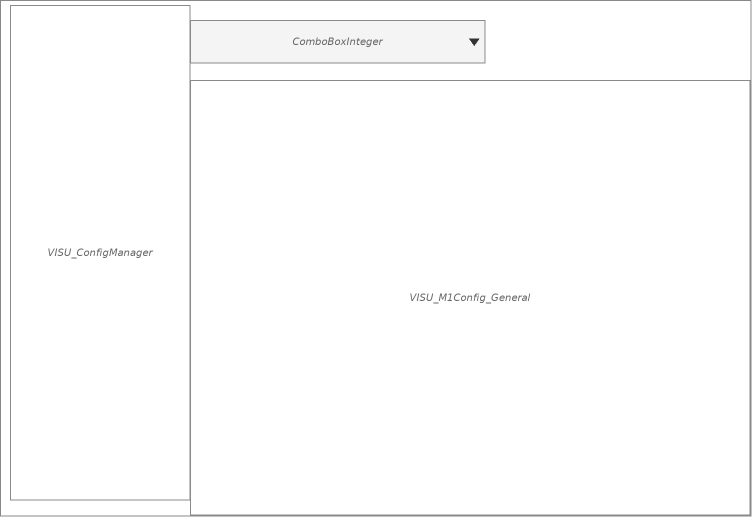
VISUALIZATION VISU_M1Config  // 752x517
VAR_IN_OUT
    editableConfig : M1Config;
	activeConfig : M1Config;
    mgr : ConfigManager;
    mgrWidget : ConfigManagerWidget;
    activeTab : INT;
END_VAR
    Frame (10,5 180x495)
        shows VISU_ConfigManager(mgr := mgr, widget := mgrWidget)
    ComboBoxInteger (190,20 295x43), variable: activeTab, text list: 'M1ConfigTabsTextList'
    Frame (190,80 560x435), frame switch variable: activeTab
        shows VISU_M1Config_General(editable := editableConfig, active := activeConfig)
        shows VISU_M1Config_Radial_General(editable := editableConfig.radialSupport, active := activeConfig.radialSupport)
        shows VISU_M1Config_Radial_RegulatorPressure(editable := editableConfig.radialSupport, active := activeConfig.radialSupport)
        shows VISU_M1Config_Radial_MirrorPressure(editable := editableConfig.radialSupport, active := activeConfig.radialSupport)
        shows VISU_M1Config_Axial_General(editable := editableConfig.axialSupport, active := activeConfig.axialSupport)
        shows VISU_M1Config_Axial_RegulatorPressure(editable := editableConfig.axialSupport, active := activeConfig.axialSupport)
        shows VISU_M1Config_Axial_MirrorPressure(editable := editableConfig.axialSupport, active := activeConfig.axialSupport)
        shows VISU_M1Config_Axial_ForceSensors(editable := editableConfig.axialSupport, active := activeConfig.axialSupport)
        shows VISU_M1Config_Axial_AverageForce(editable := editableConfig.axialSupport, active := activeConfig.axialSupport)
        shows VISU_MeasurementConfig(active := activeConfig.inclinometerVoltage, editable := editableConfig.inclinometerVoltage)
END_VISUALIZATION

(* stored: Version 1.1.0.1, ProductVersion 3.1.4019.2
   Visu VISU_M1Config: Id {09e5d830-5fd2-4512-a30d-20b6f231e528} *)
